// Mitsubishi GX Works2 project: z03   PLC: Q02/Q02H

PROGRAM MAIN
VAR
  ko : BOOL;
END_VAR
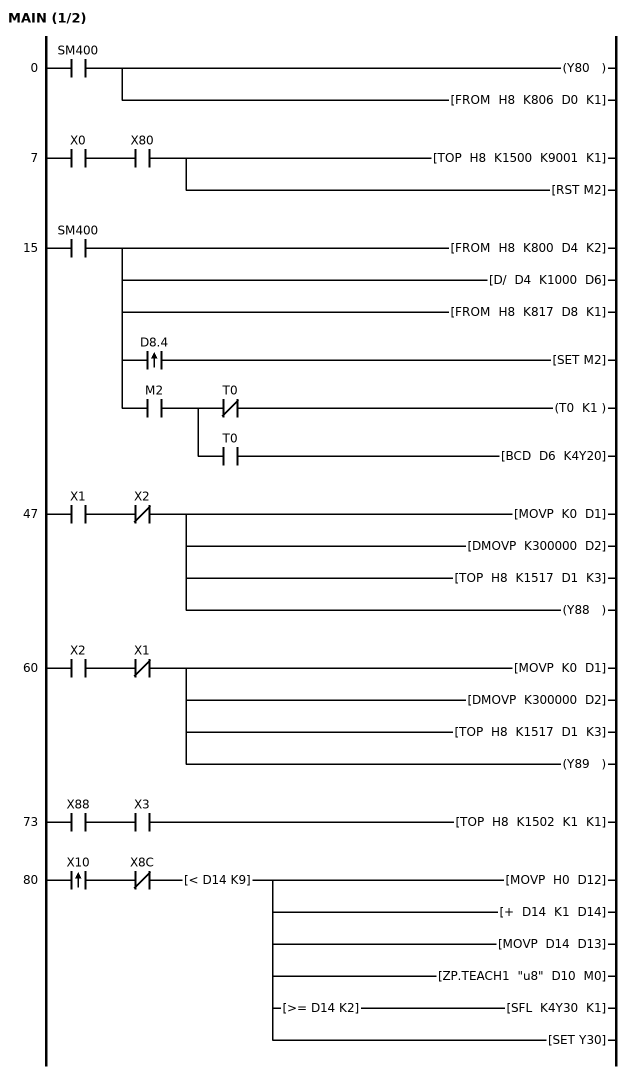
0     LD      SM400
      OUT     Y80
      FROM    H8 K806 D0 K1
7     LD      X0
      AND     X80
      TOP     H8 K1500 K9001 K1
      RST     M2
15    LD      SM400
      FROM    H8 K800 D4 K2
      D/      D4 K1000 D6
      FROM    H8 K817 D8 K1
      MPS
      ANDP    D8.4
      SET     M2
      MPP
      AND     M2
      MPS
      ANI     T0
      OUT     T0 K1
      MPP
      AND     T0
      BCD     D6 K4Y20
47    LD      X1
      ANI     X2
      MOVP    K0 D1
      DMOVP   K300000 D2
      TOP     H8 K1517 D1 K3
      OUT     Y88
60    LD      X2
      ANI     X1
      MOVP    K0 D1
      DMOVP   K300000 D2
      TOP     H8 K1517 D1 K3
      OUT     Y89
73    LD      X88
      AND     X3
      TOP     H8 K1502 K1 K1
80    LDP     X10
      ANI     X8C
      AND<    D14 K9
      MOVP    H0 D12
      +       D14 K1 D14
      MOVP    D14 D13
      ZP.TEACH1 "u8" D10 M0
      MPS
      AND>=   D14 K2
      SFL     K4Y30 K1
      MPP
      SET     Y30
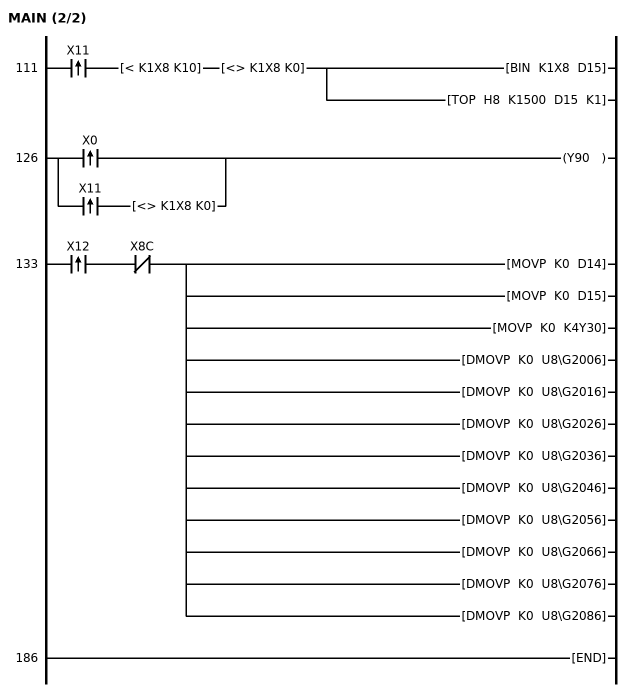
111   LDP     X11
      AND<    K1X8 K10
      AND<>   K1X8 K0
      BIN     K1X8 D15
      TOP     H8 K1500 D15 K1
126   LDP     X0
      LDP     X11
      AND<>   K1X8 K0
      ORB
      OUT     Y90
133   LDP     X12
      ANI     X8C
      MOVP    K0 D14
      MOVP    K0 D15
      MOVP    K0 K4Y30
      DMOVP   K0 U8\G2006
      DMOVP   K0 U8\G2016
      DMOVP   K0 U8\G2026
      DMOVP   K0 U8\G2036
      DMOVP   K0 U8\G2046
      DMOVP   K0 U8\G2056
      DMOVP   K0 U8\G2066
      DMOVP   K0 U8\G2076
      DMOVP   K0 U8\G2086
186   END
END_PROGRAM
